// TIA Portal V17 export
// export: Created 2025-01-08T13:55:33.7149022Z, ExportSetting WithDefaults, DisplayName Totally Integrated Automation Portal, DisplayVersion V17, DisplayName TIA Portal Openness, DisplayVersion V17, DisplayName TIA Portal Version Control Interface, DisplayVersion V17, DisplayName SINAMICS Startdrive Advanced, DisplayVersion V17 Update2, DisplayName SINAMICS Startdrive G130, G150, S120, S150, SINAMICS MV, S210, DisplayVersion V17 Update2, DisplayName SINAMICS Startdrive G110M, G120, G120C, G120D, G120P, G115D, DisplayVersion V17 Update2, DisplayName STEP 7 Professional, DisplayVersion V17, DisplayName STEP 7 Safety, DisplayVersion V17, DisplayName WinCC Advanced, DisplayVersion V17
DATA_BLOCK "DB - HSM"   // DB18
{ S7_Optimized_Access := 'FALSE' }
VERSION : 0.1
// stored: AutoNumber true, DBAccessibleFromOPCUA true, DBAccessibleFromWebserver true, IsOnlyStoredInLoadMemory false, IsWriteProtectedInAS false
   VAR RETAIN
      HSM_Side : "typeFromHMI";
      HSM_Zon1 : "typeFromHMI";
      HSM_Zon2_SideTaxStamp : "typeFromHMI";
      xDisable_Parameter_Update_HSM_Side : Bool;   // Disable update parameter changes
      xDisable_Parameter_Update_HSM_Zon1 : Bool;   // Disable update parameter changes
      xDisable_Parameter_Update_HSM_Zon2 : Bool;   // Disable update parameter changes
   END_VAR
BEGIN
   HSM_Side.rLabel_Speed := 28.0;
   HSM_Side.xBtn_Save_Par := false;
   HSM_Side.xHSM_Active := TRUE;
   HSM_Side.xGet_Parameters := false;
   HSM_Side.iLabels_Per_Trigger := 1;
   HSM_Side.iTrigger_Supression := 0;
   HSM_Side.iProduct_Sensor_Polarity := 3;
   HSM_Side.iDouble_Label := 0;
   HSM_Side.iSpeed_Int_Ext := 1;
   HSM_Side.iLabel_Length := 0;
   HSM_Side.rLabel_Position := 1.0;
   HSM_Side.rTrig_Delay := 0.0;
   HSM_Side.rSpeed_Offset := 0.0;
   HSM_Side.rGap_Sensor_To_Dispenser_Tongue := 245.0;
   HSM_Side.rLabel_Spacing := 2.0;
   HSM_Side.rPre_Dispensing_Lenght := 0.0;
   HSM_Side.rLabel_Gap := 0.0;
   HSM_Side.ConfigAndMachineParaMask.HSMConfig_1.iDesiredInternalSpeed := true;
   HSM_Side.ConfigAndMachineParaMask.HSMConfig_1.iDispenseDelay := true;
   HSM_Side.ConfigAndMachineParaMask.HSMMachine_2.iSyncOutputDelay := true;
   HSM_Side.ConfigAndMachineParaMask.HSMMachine_2.iSyncOutputLenght := true;
   HSM_Zon1.rLabel_Speed := 28.0;
   HSM_Zon1.xHSM_Active := TRUE;
   HSM_Zon1.iLabels_Per_Trigger := 1;
   HSM_Zon1.iTrigger_Supression := 0;
   HSM_Zon1.iProduct_Sensor_Polarity := 2;
   HSM_Zon1.iDouble_Label := 0;
   HSM_Zon1.iSpeed_Int_Ext := 1;
   HSM_Zon1.iLabel_Length := 0;
   HSM_Zon1.rLabel_Position := 1.0;
   HSM_Zon1.rTrig_Delay := 0.0;
   HSM_Zon1.rSpeed_Offset := 0.0;
   HSM_Zon1.rGap_Sensor_To_Dispenser_Tongue := 125.0;
   HSM_Zon1.rLabel_Spacing := 2.0;
   HSM_Zon1.rPre_Dispensing_Lenght := 0.0;
   HSM_Zon1.rLabel_Gap := 0.0;
   HSM_Zon1.ConfigAndMachineParaMask.HSMConfig_1.iDesiredInternalSpeed := true;
   HSM_Zon1.ConfigAndMachineParaMask.HSMConfig_1.iDispenseDelay := true;
   HSM_Zon1.ConfigAndMachineParaMask.HSMConfig_1.iLabelPosition := true;
   HSM_Zon2_SideTaxStamp.rLabel_Speed := 28.0;
   HSM_Zon2_SideTaxStamp.xBtn_Save_Par := false;
   HSM_Zon2_SideTaxStamp.xHSM_Active := TRUE;
   HSM_Zon2_SideTaxStamp.xGet_Parameters := false;
   HSM_Zon2_SideTaxStamp.iLabels_Per_Trigger := 1;
   HSM_Zon2_SideTaxStamp.iTrigger_Supression := 0;
   HSM_Zon2_SideTaxStamp.iProduct_Sensor_Polarity := 3;
   HSM_Zon2_SideTaxStamp.iDouble_Label := 0;
   HSM_Zon2_SideTaxStamp.iSpeed_Int_Ext := 1;
   HSM_Zon2_SideTaxStamp.iLabel_Length := 0;
   HSM_Zon2_SideTaxStamp.rLabel_Position := 1.0;
   HSM_Zon2_SideTaxStamp.rTrig_Delay := 0.0;
   HSM_Zon2_SideTaxStamp.rSpeed_Offset := 0.0;
   HSM_Zon2_SideTaxStamp.rGap_Sensor_To_Dispenser_Tongue := 125.0;
   HSM_Zon2_SideTaxStamp.rLabel_Spacing := 2.0;
   HSM_Zon2_SideTaxStamp.rPre_Dispensing_Lenght := 0.0;
   HSM_Zon2_SideTaxStamp.rLabel_Gap := 0.0;
   HSM_Zon2_SideTaxStamp.ConfigAndMachineParaMask.HSMConfig_1.iDesiredInternalSpeed := true;
   HSM_Zon2_SideTaxStamp.ConfigAndMachineParaMask.HSMConfig_1.iDispenseDelay := true;
   HSM_Zon2_SideTaxStamp.ConfigAndMachineParaMask.HSMConfig_1.iLabelPosition := true;
   HSM_Zon2_SideTaxStamp.ConfigAndMachineParaMask.HSMMachine_1.iDistanceToDispensingEdgeToGapSensor := true;
END_DATA_BLOCK
